Universal Robots PolyScope program: RQ_2FG_Open2.urp

ProgramRoot directory=/home/ur/ursim-1.7_UR10/programs/Robotiq/2_Finger_Adaptive_Robot_Gripper; kinematics=(a=[0, -0.612, -0.5723, 0, 0, 0], d=[0.1273, 0, 0, 0.16394, 0.1157, 0.0922], alpha=[1.5708, 0, 0, 1.5708, -1.5708, 0], deltaTheta=[0, 0, 0, 0, 0, 0], status=notInitialized); name=RQ_2FG_Open2; programVersion=(project__name=PolyScope, major__version=1, minor__version=7, svn__revision=9981, build__date=Feb 21 2013, 15:22:49); robotEnvironmentFileName=RQ_2FG_Installation
  MainProgram cartesianAcceleration=1.2; cartesianSpeed=0.25; jointAcceleration=1.3962634015954636; jointSpeed=1.0471975511965976; moveAsFastAsPossible=true; sharedProcessMoveBlendRadius=0.025; featureReference=(installationNameReference=Base); motionType=JOINT_SPACE; runOnlyOneCycle=true
    Assignment assignmentValueSource=0; expr=100; operatorValueType=INTEGER; valueSource=EXPRESSION; variable=(name=Position_open2, prefersPersistentValue=false, requestANewUniqueName=false)
    Assignment assignmentValueSource=0; expr=100; operatorValueType=INTEGER; valueSource=EXPRESSION; variable=(name=Speed_open2, prefersPersistentValue=false, requestANewUniqueName=false)
    Assignment assignmentValueSource=0; expr=100; operatorValueType=INTEGER; valueSource=EXPRESSION; variable=(name=Force_open2, prefersPersistentValue=false, requestANewUniqueName=false)
    Script type=1; cachedFileContents=#Allocation of modbus output registers with the desired settings
      | out_reg2_open = Speed_open2 * 256 + Force_open2
      | modbus_set_output_register("Speed_Force_Req", out_reg2_open, False)
      | modbus_set_output_register("Position_Req", Position_open2, False)
      | 
      | #Allow movement
      | modbus_set_output_signal("Go_to_Requested", True, False)
      | while(modbus_get_signal_status("Action_Status", False) == False):
      |     sync()
      | end
      | 
      | #Wait until the end of the movement
      | sleep(0.2)
      | while (not((modbus_get_signal_status("Obj_Det_Status1", False) == True) or (modbus_get_signal_status("Obj_Det_Status2", False) == True ))):
      |     sleep(0.1)
      |     sync()
      | end
      | 
      | sleep(0.2)
      | #Status check object detection
      | global obj_detect1 = modbus_get_signal_status("Obj_Det_Status1",False)
      | global obj_detect2 = modbus_get_signal_status("Obj_Det_Status2",False)
      | if ((obj_detect1 == False) and (obj_detect2 == True)):
      |     global Contact_opening = False
      |     global Contact_closing = True
      | else:
      |     if ((obj_detect1 == True) and (obj_detect2 == False)):
      |         global Contact_opening = True
      |         global Contact_closing = False
      |     else:
      |         global Contact_opening = False
      |         global Contact_closing = False
      |     end
      | end
      | 
      | #Prohibit the movement
      | modbus_set_output_signal("Go_to_Requested", False, False)
      | while(modbus_get_signal_status("Action_Status", False) == True):
      |     sync()
      | end; scriptFile=/home/ur/ursim-1.7_UR10/programs/Robotiq/2_Finger_Adaptive_Robot_Gripper/RQ_2FG_Open_script2.script
